FUNCTION_BLOCK EL1098
VAR
	_io : EL1xx8_Data;
	{attribute addProperty Name "WcState"}
	_wcState : WcStateInputToggle;
	{attribute addProperty Name "Info data"}
	_infoData : InfoDataBase;
END_VAR

PROPERTY IO : REFERENCE TO EL1xx8_Data
GET
IO REF= _io;
END_GET
END_PROPERTY

PROPERTY WcState : REFERENCE TO WcStateInputToggle
GET
WcState REF= _wcState;
END_GET
END_PROPERTY

END_FUNCTION_BLOCK

(* stored: Version 1.1.0.1, ProductVersion 3.1.4024.9
   POU EL1098: Id {f054be23-768e-07ec-2f56-6cf51421b85a}, SpecialFunc None
   Property IO: Id {02695b24-a382-01ca-35a0-02531134dded}
   Get Get: Id {d83d31cf-4dec-06d4-3248-f0b7bebe2c20}
   Property WcState: Id {dbbb16b4-de9a-02cb-0e80-72c0389136fe}
   Get Get: Id {5dbb9cad-be42-049f-16da-7053fc915791} *)
